INTERFACE I_Statemachine EXTENDS I_Component

METHOD ChangeState
VAR_INPUT
	StateCommand : DINT;
END_VAR
END_METHOD

{attribute 'monitoring' := 'call'}
PROPERTY CurrentState : DINT
GET
END_GET
END_PROPERTY

PROPERTY Mode : I_Mode
GET
END_GET
SET
END_SET
END_PROPERTY

PROPERTY States : I_StateList
GET
END_GET
END_PROPERTY

END_INTERFACE

(* stored: Version 1.1.0.1, ProductVersion 3.1.4026.18
   Itf I_Statemachine: Id {713d239e-6e4d-45f2-a5b8-5ea7545de62c}
   Method ChangeState: Id {392e6d81-5943-4e1b-8c3d-080bcf40649f}
   Property CurrentState: Id {3e9a7ee7-4265-4b86-afc6-b1ddf2b07526}
   Get Get: Id {33a01a45-8da2-43c1-b23f-90eeae3805bb}
   Property Mode: Id {5c08f552-bd62-478c-9a97-ac0590fd22be}
   Get Get: Id {2586ded4-a03c-4b93-a507-99d77ad8513e}
   Set Set: Id {d32270cc-db78-4ee9-8cd7-3fb607ca681a}
   Property States: Id {e120a981-b54a-4cc9-b7bf-c85fe0c63b4f}
   Get Get: Id {6a22d756-50e5-4243-b35f-e5df0f125004} *)
